{attribute 'GeneratedUsingTerminal: EP1122-0001-0017'}
{attribute addProperty BoxType "EP1122-0001-0017"}
{attribute addProperty Id "A_0026_EP1122_0001_0018A_0026_EP1122_0001_0018_73CBC47E1450"}
{attribute addProperty CRC "1231960630"}
{attribute addProperty Size "1450"}
TYPE A_0025_EP1122_0001_0017_496E3A36 EXTENDS EP1122_1FC0878B :
STRUCT
	{attribute addProperty Name "A_0026(EP1122-0001-0018)"}
	{attribute addProperty PreviousPort "A_0025(EP1122-0001-0017) : D"}
	A_0026_EP1122_0001_0018 : A_0026_EP1122_0001_0018_73CBC47E;
END_STRUCT
END_TYPE

(* stored: Version 1.2.0.0, ProductVersion 3.1.4024.9
   DUT A_0025_EP1122_0001_0017_496E3A36: Id {1d6aa7ea-4a82-409f-9440-1e68f2cbecbb} *)
